FUNCTION_BLOCK CM_Valve IMPLEMENTS  ITF_Valve2
VAR
	fb_mem : STRUCT_CM_Valve;
END_VAR

(*
$$$$$$$$\                                                                   $$\       $$$$$$$$\                     $$\                                         $$\                     
$$  _____|                                                                  $$ |      $$  _____|                    \__|                                        \__|                    
$$ |   $$$$$$\   $$$$$$\  $$$$$$$\  $$\  $$\  $$\  $$$$$$\   $$$$$$\   $$$$$$$ |      $$ |      $$$$$$$\   $$$$$$\  $$\ $$$$$$$\   $$$$$$\   $$$$$$\   $$$$$$\  $$\ $$$$$$$\   $$$$$$\  
$$$$$\ \____$$\ $$  __$$\ $$  __$$\ $$ | $$ | $$ |$$  __$$\ $$  __$$\ $$  __$$ |      $$$$$\    $$  __$$\ $$  __$$\ $$ |$$  __$$\ $$  __$$\ $$  __$$\ $$  __$$\ $$ |$$  __$$\ $$  __$$\ 
$$  __|$$$$$$$ |$$ |  \__|$$ |  $$ |$$ | $$ | $$ |$$ /  $$ |$$ /  $$ |$$ /  $$ |      $$  __|   $$ |  $$ |$$ /  $$ |$$ |$$ |  $$ |$$$$$$$$ |$$$$$$$$ |$$ |  \__|$$ |$$ |  $$ |$$ /  $$ |
$$ |  $$  __$$ |$$ |      $$ |  $$ |$$ | $$ | $$ |$$ |  $$ |$$ |  $$ |$$ |  $$ |      $$ |      $$ |  $$ |$$ |  $$ |$$ |$$ |  $$ |$$   ____|$$   ____|$$ |      $$ |$$ |  $$ |$$ |  $$ |
$$ |  \$$$$$$$ |$$ |      $$ |  $$ |\$$$$$\$$$$  |\$$$$$$  |\$$$$$$  |\$$$$$$$ |      $$$$$$$$\ $$ |  $$ |\$$$$$$$ |$$ |$$ |  $$ |\$$$$$$$\ \$$$$$$$\ $$ |      $$ |$$ |  $$ |\$$$$$$$ |
\__|   \_______|\__|      \__|  \__| \_____\____/  \______/  \______/  \_______|      \________|\__|  \__| \____$$ |\__|\__|  \__| \_______| \_______|\__|      \__|\__|  \__| \____$$ |
                                                                                                          $$\   $$ |                                                          $$\   $$ |
      			                                                                                          \$$$$$$  |                                                          \$$$$$$  |
                                                                                                           \______/                                                            \______/ 
*)
fb_mem.STS.State := PackML_StateMachine(State			:= fb_mem.STS.State,
										Start           := fb_mem.CS.Start,
										Stop            := fb_mem.CS.Stop,
										Reset           := fb_mem.CS.Reset,
										Abort           := fb_mem.CS.Abort,
										Clear           := fb_mem.CS.Clear,
										UnSuspend       := fb_mem.CS.UnSuspend,
										Suspend         := fb_mem.CS.Suspend,
										UnHold          := fb_mem.CS.UnHold,
										Hold            := fb_mem.CS.Hold,
										Starting_SC     := fb_mem.STS.Starting_SC,
										Execute_SC      := fb_mem.STS.Execute_SC,
										Completing_SC	:= fb_mem.STS.Completing_SC,
										Resetting_SC    := fb_mem.STS.Resetting_SC,
										Holding_SC      := fb_mem.STS.Holding_SC,
										Unholding_SC    := fb_mem.STS.Unholding_SC,
										Suspending_SC   := fb_mem.STS.Suspending_SC,
										Unsuspending_SC := fb_mem.STS.Unsuspending_SC,
										Aborting_SC     := fb_mem.STS.Aborting_SC,
										Clearing_SC     := fb_mem.STS.Clearing_SC,
										Stopping_SC     := fb_mem.STS.Stopping_SC);

//********************************Auto manual logic***********************************
IF fb_mem.CS.Auto OR fb_mem.HMI.Auto THEN
	fb_mem.STS.Auto := TRUE;
	fb_mem.STS.Manueel := FALSE;
END_IF

IF fb_mem.CS.Manueel OR fb_mem.HMI.Manueel THEN
	fb_mem.STS.Auto := FALSE;
	fb_mem.STS.Manueel := TRUE;
END_IF

//********************************Exeptionhandling***********************************

//********************************Action case***********************************
CASE fb_mem.STS.State OF
	E_State_PackML.IDLE 			:
		//Do nothing
	E_State_PackML.STARTING 		:
		fb_mem.STS.Starting_SC 		:= TRUE;
	E_State_PackML.EXECUTE 			: 
		//Do nothing
	E_State_PackML.COMPLETING		:
		fb_mem.STS.Completing_SC := TRUE;
	E_State_PackML.COMPLETE 		:
		IF fb_mem.CS.Clear AND fb_mem.STS.Auto OR fb_mem.HMI.Clear AND fb_mem.STS.Manueel THEN
			fb_mem.STS.Completing_SC := TRUE;
		END_IF
	E_State_PackML.RESETTING 		:
		FB_init(0,0);
		fb_mem.STS.Resetting_SC 	:= TRUE;
	E_State_PackML.HOLDING 			:
		fb_mem.STS.Unholding_SC		:= TRUE;
	E_State_PackML.HELD 			:
		//Do nothing
	E_State_PackML.UNHOLDING 		:
		fb_mem.STS.Unholding_SC		:= TRUE;
	E_State_PackML.SUSPENDING 		:
		fb_mem.STS.Suspending_SC 	:= TRUE;
	E_State_PackML.SUSPENDED 		:
		fb_mem.CS.Unsuspend 		:= TRUE;
	E_State_PackML.UNSUSPENDING 	:
		fb_mem.STS.Unsuspending_SC 	:= TRUE;
	E_State_PackML.ABORTED			:
		//Do nothing
	E_State_PackML.ABORTING			:
		fb_mem.STS.Aborting_SC 		:= TRUE;
	E_State_PackML.CLEARING 		:
		fb_mem.STS.Clearing_SC 		:= TRUE;
	E_State_PackML.STOPPING 		:
		fb_mem.STS.Stopping_SC 		:= TRUE;
	E_State_PackML.STOPPED 			:
		//Do nothing
		
END_CASE




//Zero all CS signals
fb_mem.CS.Auto			:= FALSE;
fb_mem.CS.Manueel 		:= FALSE;
fb_mem.CS.Abort			:= FALSE;
fb_mem.CS.Reset			:= FALSE;
fb_mem.CS.Start			:= FALSE;
fb_mem.CS.Stop			:= FALSE;

//Zero all HMI signals
fb_mem.HMI.Auto			:= FALSE;
fb_mem.HMI.Manueel 		:= FALSE;
fb_mem.HMI.Abort		:= FALSE;
fb_mem.HMI.Reset		:= FALSE;
fb_mem.HMI.Start		:= FALSE;
fb_mem.HMI.Stop			:= FALSE;

{warning 'add method implementation '}
METHOD Abort : BOOL
fb_mem.CS.Abort := TRUE;

Abort := fb_mem.CS.Abort;
END_METHOD

PROPERTY Auto : BOOl
GET
AUTO := fb_mem.STS.Auto;
END_GET
SET
fb_mem.CS.Auto := AUTO;
END_SET
END_PROPERTY

METHOD Clear : BOOL
VAR_INPUT
END_VAR
fb_mem.CS.Clear := TRUE;

Clear := fb_mem.CS.Abort;
END_METHOD

{warning 'add method implementation '}
METHOD Close : BOOL
fb_mem.CS.Close := TRUE;
fb_mem.STS.Close:=TRUE;
fb_mem.STS.Open:=FALSE;
Close := fb_mem.STS.Close;
END_METHOD

{warning 'add property implementation'}
PROPERTY Error_State : E_Motor_Error_State
GET
Error_State := fb_mem.STS.Error_State;
END_GET
END_PROPERTY

METHOD FB_init : BOOL
VAR_INPUT
	bInitRetains : BOOL; // if TRUE, the retain variables are initialized (warm start / cold start)
	bInCopyCode : BOOL;  // if TRUE, the instance afterwards gets moved into the copy code (online change)
END_VAR
fb_mem.STS.State := E_State_PackML.IDLE;
END_METHOD

PROPERTY Manueel : BOOl
GET
Manueel := fb_mem.STS.Manueel;
END_GET
SET
fb_mem.CS.Manueel :=  Manueel;
END_SET
END_PROPERTY

{warning 'add method implementation '}
METHOD Open : BOOL
fb_mem.CS.Open := TRUE;
fb_mem.STS.Open:=TRUE;
fb_mem.STS.Close:=FALSE;
Open := fb_mem.STS.Open;
END_METHOD

{warning 'add method implementation '}
METHOD Reset : BOOL
fb_mem.CS.Reset := TRUE;

Reset := fb_mem.CS.Reset;
END_METHOD

{warning 'add method implementation '}
METHOD Start : BOOL
fb_mem.CS.Start := TRUE;

Start := fb_mem.CS.Start;
END_METHOD

{warning 'add property implementation'}
PROPERTY State : E_Motor_State
GET
END_GET
END_PROPERTY

{warning 'add method implementation '}
METHOD Stop : BOOL
fb_mem.CS.Stop := TRUE;

Stop := fb_mem.CS.Stop;
END_METHOD

PROPERTY Tag : STRING
GET
Tag := fb_mem.STS.Tag;
END_GET
END_PROPERTY

END_FUNCTION_BLOCK

(* stored: Version 1.1.0.1, ProductVersion 3.1.4024.12
   POU CM_Valve: Id {50d84cc6-aa4d-44df-b18f-022b3ce5e0ef}, SpecialFunc None
   Folder Methods: Id {e46b56ed-db35-46c1-8cab-d3ea75e448a6}
   Folder Properties: Id {051e65f6-b3f6-4d6d-ad1b-b059338e4c4c}
   Method Abort: Id {6bba516f-ae66-4e07-a358-2d89a647406e}
   Property Auto: Id {23207d80-76f5-4441-978d-04010994bcd9}
   Get Get: Id {ca848de0-4684-4a3c-b25b-1cf8887283a3}
   Set Set: Id {4df17699-961e-45f2-a912-bdefcf8b1afc}
   Method Clear: Id {5b15b59a-be31-472b-9d4e-65c002739a05}
   Method Close: Id {f05bfdcd-7296-4824-890e-d5f7a842ca33}
   Property Error_State: Id {dc8aa90f-9928-4995-8038-ee1ec047b629}
   Get Get: Id {672153e2-6096-473a-81c2-7ada8a12d856}
   Method FB_init: Id {5c4fd80b-892a-43fc-9bf4-2daff6db55bf}
   Property Manueel: Id {e8fef718-509b-4976-add4-66d742661a2f}
   Get Get: Id {12df9233-0666-4ea0-8ad6-4a5550edf652}
   Set Set: Id {2ee474ea-1eb2-481c-b217-f0c945709a76}
   Method Open: Id {2d5e1512-428d-4d24-b750-a85ea72d1fde}
   Method Reset: Id {e7cf8f8d-ac8a-43e7-9347-40ccade0c41d}
   Method Start: Id {a2d1ea15-ee1f-4e23-bec2-fa9d84a753a5}
   Property State: Id {a759bc80-5e36-4408-88d3-cfd6503a2bbf}
   Get Get: Id {8f60474b-c8f5-4540-910a-259f36868ab6}
   Method Stop: Id {69145ac8-7c54-4ce2-8357-436d1f812573}
   Property Tag: Id {cfe256b7-2fd2-4ea5-ad89-2952dcc0d2e2}
   Get Get: Id {409b834e-8f90-41b6-9348-0a6f5679bccf} *)
